{attribute 'qualified_only'}
{attribute 'strict'}
TYPE eCommandTypes :
(
	NO_OPERATION := 0,
	POSITION:=1,
	ZRET:=3,
	
	SET_POSITION:=16#FF
);
END_TYPE

(* stored: Version 1.1.0.1, ProductVersion 3.1.4022.10
   DUT eCommandTypes: Id {fa388b91-8966-4e52-bc41-23d3150b895c} *)
